# B&R Automation Studio project program bez kamery
Automation Studio 4.9

## Configuration Config1

CPU 5APC3100.KBU1-000, AutomationRuntime J4.93, Build 4.1.2, Safety 0.0, Vc V4.73.2

CPU 5APC3100.KBU1-000, AutomationRuntime J4.93, Build 4.1.2, Safety 0.0, Vc V4.73.2

### Task classes (Cpu.sw)
```
Cyclic#1:
  PrgMechs <- PickAndPlace.PrgMechs.prg
  PrgPickCor <- PickAndPlace.PrgPickCore.prg
  PrgPick <- PickAndPlace.PrgPick.prg
  PrgPlace <- PickAndPlace.PrgPlace.prg
DataObjects: McAcpSys
NcDataObjects: McDriveLog
Binaries: McAcpDrv, udbdef, McAcpSim, mvLoader, arflatprv, TCData, McProfGen, mCoWebSc, McMechSys, FWRules, arcoal, arsvcreg, Settings, iomap, Config_3, Config_4, Role, ashwac, Config_10, asfw, Config_5, sysconf, Config_2, arconfig, Config_6, Config_8, Config_1, Hierarchy, ashwd, Config_7, User, Config_9
Libraries: UserLib, McBase, MpBase, MpRobotics, McAxGroup, McPathGen, McAxis, McProgInt, McAcpAx, CoTrace, AsZip, FileIO, runtime, MpAxis, McAcpPar, McTrkPath, MpPick, McAcpTrak, MpCnc, MpTool, sys_lib, McDS402Ax, McPureVAx, McStpAx, asarprof, asarlog, asio, asmem, astime, asepl, dataobj, brsystem, arssl, powerlnk, asioacc, asieccon
```

### Task classes (Cpu.sw)
```
Libraries: McBase, MpBase, McAcpAx, McAxis, McAcpPar, McAxGroup, McDS402Ax, McPureVAx, McStpAx, McPathGen, McProgInt, McTrkPath, MpPick, McAcpTrak, MpAxis, MpCnc, MpRobotics, MpTool, sys_lib, runtime
```

### Config_4.axesgroupfeature - 5APC3100_KBU1_000a/mappMotion/4AxesDeltaA/Config_4.axesgroupfeature
```
Element Feature_Programs (Type=axesgroupfeature)
  Type = Program
    ModalDataBehaviour = UseAxesGroupSettings
    InitialSettings:
      InterpolationTypes = LinearRapid
      PositionCoordinates = Absolute
      CircleCoordinates = Relative
      JACS_ACSProgramming = JACS
      ContourConnection = Inactive
      ProgrammingUnits = UseAxesGroupSettings
      Feedrates:
        FeedPath = Standard
        FeedCharacteristic = StandardCharacteristic
        FeedType = Feedrate
        FeedReduction = Inactive
        FeedrateValue = 0.0
        InverseFeedrateValue = 0.0
        FeedratePerRevValue = 0.0
    DefaultLanguage = BRGCode
    Location = Default
      FileDevice = CNC_PrgDir
Element Feature_Jogging (Type=axesgroupfeature)
  Type = Jogging
Element Feature_MotionPacketLog (Type=axesgroupfeature)
  Type = MotionPacketLog
    Location = User
      FileDevice = CNC_PrgDir
```

### Config_6.axesgroupfeature - 5APC3100_KBU1_000a/mappMotion/PnP_AddOn/Config_6.axesgroupfeature
```
Element Feature_FrameHierarchy (Type=axesgroupfeature)
  Type = FrameHierarchy
    ModalDataBehaviour = UseAxesGroupSettings
    FrameHierarchy = Custom
      FramePropertyMapping:
        BCS = RoboBase
        PCS = ZeroPosPickConveyor
        SCS1
        SCS2
        SCS3
        SCS4
        SCS5
      MCS:
        Name = MachineBase
        Frame[1]:
          Name = RoboBase
          Type = StandardFrame
            Translation:
              X = 0.0
              Y = 0
              Z = 490
            Orientation:
              Angle1 = 0.0
              Angle2 = 0.0
              Angle3 = 0.0
          Frame[1]:
            Name = ZeroPosPickConveyor
            Type = StandardFrame
              Translation:
                X = -300
                Y = 0
                Z = -430
              Orientation:
                Angle1 = 0.0
                Angle2 = 0.0
                Angle3 = 0.0
Element Feature_Tracking (Type=axesgroupfeature)
  Type = Tracking
    ModalDataBehaviour = UseAxesGroupSettings
    SynchronisationGeometry = Basic
      CartesianRadius = 20.0
    TorqueLimitConsideration = Exact
Element Feature_PathDefinition (Type=axesgroupfeature)
  Type = PathDefinitions
    ModalDataBehaviour = UseAxesGroupSettings
    PathDefinition[1]:
      Name = Path1
      Type = CartesianPath
        CalculatedIn = PCS
      Limit = Internal
        Velocity = NotUsed
        Acceleration = NotUsed
        Deceleration = NotUsed
        Jerk = NotUsed
```

### Config_8.pickregister - 5APC3100_KBU1_000a/mappMotion/PnP_AddOn/Config_8.pickregister
```
Element gPickRegister (Type=pickregister)
  Type = LinearConveyor
    StandardFrameName = ConveyorPick
    Length = 600
    Width = 120
    Height = 10
    MotionSource = Axis
      AxisRef = gAxis_1
      MovementLimits = UseAxisLimits
  SceneViewerObject = Used
    VisualRepresentation = Conveyor belt
      Dimensions:
        Length = 610
        Width = 120
        Height = 50
      Translation:
        X = 0
        Y = 0.0
        Z = 0.0
      Orientation:
        Angle1 = 0.0
        Angle2 = 0.0
        Angle3 = 0.0
      Material = GreenMatte
    Content:
      Template[1]:
        VisualRepresentation = 2DShape
          ShapeType:
            Dimensions:
              Radius = 25.0
            Translation:
              X = 0.0
              Y = 0.0
              Z = 0
            Orientation:
              Angle1 = 0.0
              Angle2 = 0.0
              Angle3 = 0.0
        Filter:
          ObjectState:
            State[1] = 1
      Template[2]:
        VisualRepresentation:
          Size = 50.0
        Filter:
          ObjectState:
            State[1] = 2
  Alarms = None
Element gPlaceRegister (Type=pickregister)
  Type = LinearConveyor
    StandardFrameName = ConveyorPlace
    Length = 205
    Width = 60
    Height = 10
    MaxItems = 5
    MotionSource = Axis
      AxisRef = gAxis_2
      MovementLimits = UseAxisLimits
  SceneViewerObject = Used
    Dimensions:
      Material = Undefined
    VisualRepresentation = Cuboid
      Dimensions:
        Length = 215
        Width = 60
        Height = 50
      Translation:
        X = 0
        Y = 0
        Z = 0.0
      Orientation:
        Angle1 = 0.0
        Angle2 = 0.0
        Angle3 = 0.0
    Content:
      Template[1]:
        VisualRepresentation = 2DShape
          ShapeType:
            Dimensions:
              Radius = 25.0
            Translation:
              X = 0.0
              Y = 0.0
              Z = 0.0
            Orientation:
              Angle1 = 0.0
              Angle2 = 0.0
              Angle3 = 0.0
        Filter:
          ObjectState:
            State[1] = 7
      Template[2]:
        VisualRepresentation:
          Size = 50.0
        Filter:
          ObjectState:
            State[1] = 2
  Alarms = None
```

### Config_2.axis - PC/mappMotion/4AxesDeltaA/Config_2.axis
```
Element gAxisQ1 (Type=axis)
  BaseTypeIsReadOnly = 0
  BaseType = RotaryBounded
    MeasurementUnitIsReadOnly = 0
    MeasurementUnit = 17476
    MeasurementResolutionIsReadOnly = 0
    MeasurementResolution = 0.01
    CountDirectionIsReadOnly = 0
    CountDirection = Standard
  MovementLimitsIsReadOnly = 0
  MovementLimits = Internal
    Position:
      LowerLimitMin = -1.79769313486231E308
      UpperLimitMax = 1.79769313486231E308
      LowerLimit = -1000.0
      UpperLimit = 1000.0
    VelocityIsReadOnly = 0
    Velocity:
      VelocityMax = 3.4E38
      Velocity = 10.0
    AccelerationIsReadOnly = 0
    Acceleration:
      AccelerationMax = 3.4E38
      Acceleration = 50.0
    DecelerationIsReadOnly = 0
    Deceleration:
      DecelerationMax = 3.4E38
      Deceleration = 50.0
  Alarms = None
Element gAxisQ2 (Type=axis)
  BaseTypeIsReadOnly = 0
  BaseType = RotaryBounded
    MeasurementUnitIsReadOnly = 0
    MeasurementUnit = 17476
    MeasurementResolutionIsReadOnly = 0
    MeasurementResolution = 0.01
    CountDirectionIsReadOnly = 0
    CountDirection = Standard
  MovementLimitsIsReadOnly = 0
  MovementLimits = Internal
    Position:
      LowerLimitMin = -1.79769313486231E308
      UpperLimitMax = 1.79769313486231E308
      LowerLimit = -1000.0
      UpperLimit = 1000.0
    VelocityIsReadOnly = 0
    Velocity:
      VelocityMax = 3.4E38
      Velocity = 10.0
    AccelerationIsReadOnly = 0
    Acceleration:
      AccelerationMax = 3.4E38
      Acceleration = 50.0
    DecelerationIsReadOnly = 0
    Deceleration:
      DecelerationMax = 3.4E38
      Deceleration = 50.0
  Alarms = None
Element gAxisQ3 (Type=axis)
  BaseTypeIsReadOnly = 0
  BaseType = RotaryBounded
    MeasurementUnitIsReadOnly = 0
    MeasurementUnit = 17476
    MeasurementResolutionIsReadOnly = 0
    MeasurementResolution = 0.01
    CountDirectionIsReadOnly = 0
    CountDirection = Standard
  MovementLimitsIsReadOnly = 0
  MovementLimits = Internal
    Position:
      LowerLimitMin = -1.79769313486231E308
      UpperLimitMax = 1.79769313486231E308
      LowerLimit = -1000.0
      UpperLimit = 1000.0
    VelocityIsReadOnly = 0
    Velocity:
      VelocityMax = 3.4E38
      Velocity = 10.0
    AccelerationIsReadOnly = 0
    Acceleration:
      AccelerationMax = 3.4E38
      Acceleration = 50.0
    DecelerationIsReadOnly = 0
    Deceleration:
      DecelerationMax = 3.4E38
      Deceleration = 50.0
  Alarms = None
Element gAxisQ4 (Type=axis)
  BaseTypeIsReadOnly = 0
  BaseType = RotaryBounded
    MeasurementUnitIsReadOnly = 0
    MeasurementUnit = 17476
    MeasurementResolutionIsReadOnly = 0
    MeasurementResolution = 0.01
    CountDirectionIsReadOnly = 0
    CountDirection = Standard
  MovementLimitsIsReadOnly = 0
  MovementLimits = Internal
    Position:
      LowerLimitMin = -1.79769313486231E308
      UpperLimitMax = 1.79769313486231E308
      LowerLimit = -1000.0
      UpperLimit = 1000.0
    VelocityIsReadOnly = 0
    Velocity:
      VelocityMax = 3.4E38
      Velocity = 10.0
    AccelerationIsReadOnly = 0
    Acceleration:
      AccelerationMax = 3.4E38
      Acceleration = 50.0
    DecelerationIsReadOnly = 0
    Deceleration:
      DecelerationMax = 3.4E38
      Deceleration = 50.0
  Alarms = None
```

### Config_3.mechanicalsystem - PC/mappMotion/4AxesDeltaA/Config_3.mechanicalsystem
```
Element MechSys_4AxDeltaA (Type=mechanicalsystem)
  TypeIsReadOnly = 0
  Type = Delta
    SubtypeIsReadOnly = 0
    Subtype = 4AxesDeltaA
      SceneViewerObject = Generic
      DescriptionIsReadOnly = 0
      Description = Standard
        Dimensions:
          BasePlatform:
            CenterIsReadOnly = 0
            Center:
              X = 310.0
              Y = 310.0
              Z = 490.0
            ArmLinkPointIsReadOnly = 0
            Arm1LinkPoint:
              Angle = -90.0
              Radius = 150.0
              Z = 0.0
            Arm2LinkPoint:
              Angle = 0.0
              Radius = 130.0
              Z = 80.0
            Arm3LinkPoint:
              Angle = 90.0
              Radius = 150.0
              Z = 0.0
          Arms:
            ArmIsReadOnly = 0
            Arm1:
              UpperArmLength = 150.0
              LowerArmLength = 430.0
            Arm2:
              UpperArmLength = 150.0
              LowerArmLength = 430.0
            Arm3:
              UpperArmLength = 150.0
              LowerArmLength = 430.0
            LowerArmPairDistance = 70.0
          EndEffectorPlatform:
            ArmLinkPointIsReadOnly = 0
            Arm1LinkPoint:
              Radius = 80.0
              Z = 0.0
            Arm2LinkPoint:
              Radius = 70.0
              Z = 0.0
            Arm3LinkPoint:
              Radius = 80.0
              Z = 0.0
            TranslationToFlangeIsReadOnly = 0
            TranslationToFlange:
              X = 0.0
              Y = 0.0
              Z = -45.0
        Offsets:
          JointAxisIsReadOnly = 0
          JointAxis[1] = 0.0
          JointAxis[2] = 0
          JointAxis[3] = 0.0
          JointAxis[4] = 0.0
        CountDirections:
          JointAxisIsReadOnly = 0
          JointAxis[1] = Inverse
          JointAxis[2] = Standard
          JointAxis[3] = Standard
          JointAxis[4] = Standard
      CoordinatesNames = Default
        XCoordinateName = X
        YCoordinateName = Y
        ZCoordinateName = Z
        CCoordinateName = C
      WireFrameModelIsReadOnly = 0
      WireFrameModel = Standard
        UpperArm1IsReadOnly = 0
        UpperArm1 = ConnectionLine
          DistanceMin = -1.79769313486231E308
          DistanceMax = 1.79769313486231E308
          Distance = 0.0
        LowerArm1IsReadOnly = 0
        LowerArm1 = ConnectionLine
          DistanceMin = -1.79769313486231E308
          DistanceMax = 1.79769313486231E308
          Distance = 0.0
        UpperArm2IsReadOnly = 0
        UpperArm2 = ConnectionLine
          DistanceMin = -1.79769313486231E308
          DistanceMax = 1.79769313486231E308
          Distance = 0.0
        LowerArm2IsReadOnly = 0
        LowerArm2 = ConnectionLine
          DistanceMin = -1.79769313486231E308
          DistanceMax = 1.79769313486231E308
          Distance = 0.0
        UpperArm3IsReadOnly = 0
        UpperArm3 = ConnectionLine
          DistanceMin = -1.79769313486231E308
          DistanceMax = 1.79769313486231E308
          Distance = 0.0
        LowerArm3IsReadOnly = 0
        LowerArm3 = ConnectionLine
          DistanceMin = -1.79769313486231E308
          DistanceMax = 1.79769313486231E308
          Distance = 0.0
        EndEffectorPlatformToFlangeIsReadOnly = 0
        EndEffectorPlatformToFlange = ConnectionLine
          DistanceMin = -1.79769313486231E308
          DistanceMax = 1.79769313486231E308
          Distance = 0.0
        FlangeToTcp = ConnectionLine
          DistanceMin = -1.79769313486231E308
          DistanceMax = 1.79769313486231E308
          Distance = 0.0
      DynamicModelIsReadOnly = 0
      DynamicModel = DynParTable
        TableRef
      InternalDynamicModelIsReadOnly = 0
      InternalDynamicModel = NotUsed
      DynamicLimits = DynParTables
        GearboxLimitsTableRef
        CrossSectionLimitsTableRef
      InternalDynamicLimits = NotUsed
      LoadDependentJerkLimitsIsReadOnly = 0
      LoadDependentJerkLimits = NotUsed
      CouplingsIsInvisible = 0
      JointAxesPositionLimits:
        JointAxisIsReadOnly = 0
        JointAxis[1] = UseAxisLimits
        JointAxis[2] = UseAxisLimits
        JointAxis[3] = UseAxisLimits
        JointAxis[4] = UseAxisLimits
      WorkingRangeIsReadOnly = 0
      WorkingRange = NotUsed
```

## Logical view

Binary libraries used (declarations not repeated): McBase, MpBase, McTrkPath, CoTrace, AsZip, FileIO, runtime, McAcpAx, McAxis, McAxGroup, McPathGen, McProgInt, MpPick, McAcpTrak, MpAxis, MpCnc, MpRobotics, MpTool, sys_lib, McAcpPar, McDS402Ax, McPureVAx, McStpAx, McAcpTrak 5.24.1, MpTool 5.24.1

### McTrkPathCfg.typ
```iecst
TYPE
	McTPTypEnum :
		( (*Type selector setting*)
		mcTPT_LIN := 0 (*Linear - Linear tracking path*)
		);
	McTPLinMotSrcEnum :
		( (*Motion source selector setting*)
		mcTPTLMS_POS_PROC_VAR := 0, (*Position process variable - Position provided by process variable*)
		mcTPTLMS_AX := 1 (*Axis - Axis*)
		);
	McTPLinMotSrcPosPVMoveLimEnum :
		( (*Movement limits selector setting*)
		mcTPTLMSPPVML_INT := 0 (*Internal - Internal definition of limits*)
		);
	McTPLMSPPVMLIVelEnum :
		( (*Velocity selector setting*)
		mcTPTLMSPPVMLIV_BASIC := 0 (*Basic -*)
		);
	McTPLMSPPVMLIVelBasicType : STRUCT (*Type mcTPTLMSPPVMLIV_BASIC settings*)
		Velocity : REAL; (*Velocity limit in any movement direction [Measurement units/s]*)
	END_STRUCT;
	McTPLMSPPVMLIVelType : STRUCT (*Limits for velocity*)
		Type : McTPLMSPPVMLIVelEnum; (*Velocity selector setting*)
		Basic : McTPLMSPPVMLIVelBasicType; (*Type mcTPTLMSPPVMLIV_BASIC settings*)
	END_STRUCT;
	McTPLMSPPVMLIAccEnum :
		( (*Acceleration selector setting*)
		mcTPTLMSPPVMLIA_BASIC := 0 (*Basic -*)
		);
	McTPLMSPPVMLIAccBasicType : STRUCT (*Type mcTPTLMSPPVMLIA_BASIC settings*)
		Acceleration : REAL; (*Acceleration limit in any movement direction [Measurement units/s²]*)
	END_STRUCT;
	McTPLMSPPVMLIAccType : STRUCT (*Limits for acceleration*)
		Type : McTPLMSPPVMLIAccEnum; (*Acceleration selector setting*)
		Basic : McTPLMSPPVMLIAccBasicType; (*Type mcTPTLMSPPVMLIA_BASIC settings*)
	END_STRUCT;
	McTPLMSPPVMLIType : STRUCT (*Type mcTPTLMSPPVML_INT settings*)
		Velocity : McTPLMSPPVMLIVelType; (*Limits for velocity*)
		Acceleration : McTPLMSPPVMLIAccType; (*Limits for acceleration*)
	END_STRUCT;
	McTPLinMotSrcPosPVMoveLimType : STRUCT (*Velocity, acceleration and deceleration limits to be considered*)
		Type : McTPLinMotSrcPosPVMoveLimEnum; (*Movement limits selector setting*)
		Internal : McTPLMSPPVMLIType; (*Type mcTPTLMSPPVML_INT settings*)
	END_STRUCT;
	McTPLinMotSrcPosPVPrepEnum :
		( (*Signal preparation selector setting*)
		mcTPTLMSPPVP_NO_PREP := 0, (*No preparation - Suitable for high quality input signals*)
		mcTPTLMSPPVP_LIN_REG := 1 (*Linear regression - Suitable for low quality input signals*)
		);
	McTPLinMotSrcPosPVPrepLinRegType : STRUCT (*Type mcTPTLMSPPVP_LIN_REG settings*)
		ConsideredSamples : DINT; (*Number of samples used for calculating the velocity [Samples]*)
		PositionDisturbance : LREAL; (*Considered magnitude of position disturbance effects [Measurement units]*)
	END_STRUCT;
	McTPLinMotSrcPosPVPrepType : STRUCT (*Preparation of the input signal from Motion source*)
		Type : McTPLinMotSrcPosPVPrepEnum; (*Signal preparation selector setting*)
		LinearRegression : McTPLinMotSrcPosPVPrepLinRegType; (*Type mcTPTLMSPPVP_LIN_REG settings*)
	END_STRUCT;
	McTPLinMotSrcPosPVType : STRUCT (*Type mcTPTLMS_POS_PROC_VAR settings*)
		ProcessVariableName : STRING[250]; (*Process variable name to get current position*)
		NegativeOverflow : LREAL; (*Positionoverflow in negative direction*)
		PositiveOverflow : LREAL; (*Positionoverflow in positive direction*)
		DelayTime : LREAL; (*Delay time of tracking path position signal for error compensation (filtering, delay of signals, ...) [s]*)
		MovementLimits : McTPLinMotSrcPosPVMoveLimType; (*Velocity, acceleration and deceleration limits to be considered*)
		Preparation : McTPLinMotSrcPosPVPrepType; (*Preparation of the input signal from Motion source*)
	END_STRUCT;
	McTPLinMotSrcAxAxUseEnum :
		( (*Axis usage selector setting*)
		mcTPTLMSAAU_ACT := 0, (*Active - The configured axis actively moves the transport system*)
		mcTPTLMSAAU_PASS := 1 (*Passive - The configured axis is used to filter the position input signal only*)
		);
	McTPLinMotSrcAxAxUseType : STRUCT (*Defines how the axis is used*)
		Type : McTPLinMotSrcAxAxUseEnum; (*Axis usage selector setting*)
	END_STRUCT;
	McTPLinMotSrcAxMoveLimEnum :
		( (*Movement limits selector setting*)
		mcTPTLMSAML_USE_AX_LIM := 0, (*Use axis limits - Internal definition of limits*)
		mcTPTLMSAML_INT := 1 (*Internal - Internal definition of limits*)
		);
	McTPLMSAMLIVelEnum :
		( (*Velocity selector setting*)
		mcTPTLMSAMLIV_BASIC := 0 (*Basic -*)
		);
	McTPLMSAMLIVelBasicType : STRUCT (*Type mcTPTLMSAMLIV_BASIC settings*)
		Velocity : REAL; (*Velocity limit in any movement direction [Measurement units/s]*)
	END_STRUCT;
	McTPLMSAMLIVelType : STRUCT (*Limits for velocity*)
		Type : McTPLMSAMLIVelEnum; (*Velocity selector setting*)
		Basic : McTPLMSAMLIVelBasicType; (*Type mcTPTLMSAMLIV_BASIC settings*)
	END_STRUCT;
	McTPLMSAMLIAccEnum :
		( (*Acceleration selector setting*)
		mcTPTLMSAMLIA_BASIC := 0 (*Basic -*)
		);
	McTPLMSAMLIAccBasicType : STRUCT (*Type mcTPTLMSAMLIA_BASIC settings*)
		Acceleration : REAL; (*Acceleration limit in any movement direction [Measurement units/s²]*)
	END_STRUCT;
	McTPLMSAMLIAccType : STRUCT (*Limits for acceleration*)
		Type : McTPLMSAMLIAccEnum; (*Acceleration selector setting*)
		Basic : McTPLMSAMLIAccBasicType; (*Type mcTPTLMSAMLIA_BASIC settings*)
	END_STRUCT;
	McTPLMSAMLIType : STRUCT (*Type mcTPTLMSAML_INT settings*)
		Velocity : McTPLMSAMLIVelType; (*Limits for velocity*)
		Acceleration : McTPLMSAMLIAccType; (*Limits for acceleration*)
	END_STRUCT;
	McTPLinMotSrcAxMoveLimType : STRUCT (*Velocity, acceleration and deceleration limits to be considered*)
		Type : McTPLinMotSrcAxMoveLimEnum; (*Movement limits selector setting*)
		Internal : McTPLMSAMLIType; (*Type mcTPTLMSAML_INT settings*)
	END_STRUCT;
	McTPLinMotSrcAxPrepEnum :
		( (*Signal preparation selector setting*)
		mcTPTLMSAP_NO_PREP := 0, (*No preparation - Suitable for high quality input signals*)
		mcTPTLMSAP_LIN_REG := 1 (*Linear regression - Suitable for low quality input signals*)
		);
	McTPLinMotSrcAxPrepLinRegType : STRUCT (*Type mcTPTLMSAP_LIN_REG settings*)
		ConsideredSamples : DINT; (*Number of samples used for calculating the velocity [Samples]*)
		PositionDisturbance : LREAL; (*Considered magnitude of position disturbance effects [Measurement units]*)
	END_STRUCT;
	McTPLinMotSrcAxPrepType : STRUCT (*Preparation of the input signal from Motion source*)
		Type : McTPLinMotSrcAxPrepEnum; (*Signal preparation selector setting*)
		LinearRegression : McTPLinMotSrcAxPrepLinRegType; (*Type mcTPTLMSAP_LIN_REG settings*)
	END_STRUCT;
	McTPLinMotSrcAxType : STRUCT (*Type mcTPTLMS_AX settings*)
		AxisReference : McCfgReferenceType; (*Name of the axis reference*)
		AxisUsage : McTPLinMotSrcAxAxUseType; (*Defines how the axis is used*)
		DelayTime : LREAL; (*Additional delay time of tracking path position signal for error compensation [s]*)
		MovementLimits : McTPLinMotSrcAxMoveLimType; (*Velocity, acceleration and deceleration limits to be considered*)
		Preparation : McTPLinMotSrcAxPrepType; (*Preparation of the input signal from Motion source*)
	END_STRUCT;
	McTPLinMotSrcType : STRUCT (*Source describing the tracking path movement*)
		Type : McTPLinMotSrcEnum; (*Motion source selector setting*)
		PositionProcessVariable : McTPLinMotSrcPosPVType; (*Type mcTPTLMS_POS_PROC_VAR settings*)
		Axis : McTPLinMotSrcAxType; (*Type mcTPTLMS_AX settings*)
	END_STRUCT;
	McTPLinType : STRUCT (*Type mcTPT_LIN settings*)
		MaxTrackingFrames : UINT; (*Maximum number of tracking frames*)
		MaxPositionError : LREAL; (*Maximal deviation between tracking frames and motion source position when considering tracking path movement limits [Measurement units]*)
		MotionSource : McTPLinMotSrcType; (*Source describing the tracking path movement*)
	END_STRUCT;
	McTPTypType : STRUCT (*Geometry of tracking path*)
		Type : McTPTypEnum; (*Type selector setting*)
		Linear : McTPLinType; (*Type mcTPT_LIN settings*)
	END_STRUCT;
	McCfgTrkPathType : STRUCT (*Main data type corresponding to McCfgTypeEnum mcCFG_TRK_PATH*)
		Type : McTPTypType; (*Geometry of tracking path*)
	END_STRUCT;
END_TYPE
```

### Types.typ
```iecst
TYPE
	ConvStepEnum :
		(
		C_WAIT_ENABLE,
		C_ENABLE_REGISTER_FB,
		C_WAIT_ENABLE_REGISTER_FB,
		C_ENABLE_REGISTER,
		C_WAIT_ENABLE_REGISTER,
		C_ENABLE_ADD_REGISTER_FBS,
		C_WAIT_ENABLE_ADD_REGISTER_FBS,
		C_WAIT_START_PROCESS,
		C_START_PROCESS,
		C_WAIT_PROCESS_STARTED,
		C_PROCESSING,
		C_ERROR
		);
END_TYPE
```

### Variables.var
```iecst
VAR
	MpPickCore_0 : MpPickCore;
	LastStep : PickCoreStepEnum;
	PC_Step : PickCoreStepEnum;
	Error : BOOL;
	Gripper : BOOL;
END_VAR
```

### Types.typ
```iecst
TYPE
	PlaceStepEnum :
		(
		P_WAIT_ENABLE,
		P_ENABLE_REGISTER_FB,
		P_WAIT_ENABLE_REGISTER_FB,
		P_ENABLE_REGISTER_COMP,
		P_WAIT_ENABLE_REGISTER_COMP,
		P_ENABLE_ADD_REGISTER_FBS,
		P_WAIT_ENABLE_ADD_REGISTER_FBS,
		P_WAIT_START_PROCESS,
		P_CREATE_OBJECTS,
		P_WAIT_CREATE_OBJECTS,
		P_WAIT_REGISTER_FULL,
		P_DELAY_DELETE,
		P_DELETE_OBJECTS,
		P_WAIT_DELETE_OBJECTS,
		P_DELAY_CREATE,
		P_ERROR
		);
END_TYPE
```

### Library Logical/PickAndPlace/UserLibraries/UserLib (IEC) - Service library for application

#### UserLib.st
```iecst
FUNCTION DistanceOverPeriod
    (*
       Assuming:
       Pos1 = current belt position
       Pos2 = previous belt position
       Belt rotation is monodirectional

       a more computationally efficient implementation would be : DistanceOverPeriod := (Pos1 - Pos2) MOD Period;
       but, in this way, in case of Pos1 = Pos2 DistanceOverPeriod would be 0.

       With the following implementation instead, in case of Pos1 = Pos2, DistanceOverPeriod would be = Period.

       We prefer this implementation since we assume that in case of two equal positions, most likely, a full period was passed instead of no distance at all
    *)

    IF (Pos1 > Pos2) THEN
        DistanceOverPeriod := Pos1 - Pos2;
    ELSE
        DistanceOverPeriod := Period - (Pos2 - Pos1);
    END_IF

    RETURN;

END_FUNCTION
```

Listed in the project but not available here: Logical/PickAndPlace/UserLibraries/UserLib/Types.typ, Logical/PickAndPlace/UserLibraries/UserLib/Constants.var, Logical/PickAndPlace/UserLibraries/UserLib/UserLib.fun
